Yaskawa INFORM job: S1-MOV.JBI

/JOB
//NAME S1-MOV
//POS
///NPOS 0,0,4,0,0,0
///TOOL 0
///POSTYPE PULSE
///PULSE
EC00000=-28898,221232
EC00001=70924,108240
EC00002=-83889,279840
EC00003=-4514,17248
//INST
///DATE 2023/02/06 16:42
///ATTR SC,RW
///GROUP1 ST1
NOP
MOVJ EC00000 VJ=10.00
MOVJ EC00001 VJ=10.00
MOVJ EC00002 VJ=10.00
MOVJ EC00003 VJ=10.00
END
